FUNCTION_BLOCK ABSTRACT OpticalPowermeterBase EXTENDS TExecution IMPLEMENTS IDevice
VAR_INPUT
END_VAR
VAR_OUTPUT
END_VAR
VAR
	{attribute 'OPC.UA.DA' := '0'}
	_name : STRING;
	{attribute 'OPC.UA.DA' := '0'}
	_deviceID : STRING;					
	{attribute 'OPC.UA.DA' := '0'}
	_family : DeviceFamily;	
	{attribute 'OPC.UA.DA' := '0'}
	_logger : Logger;
	{attribute 'OPC.UA.DA' := '0'}
	_message : StringBuilder;
	{attribute 'OPC.UA.DA' := '0'}
	_opticalPowermeterConfig : DeviceConfiguration;	
END_VAR

PROPERTY DeviceID : STRING
GET
DeviceID := _deviceID;
END_GET
SET
_deviceID := DeviceID;
END_SET
END_PROPERTY

PROPERTY Family : DeviceFamily
GET
Family := _family;
END_GET
SET
_family := Family;
END_SET
END_PROPERTY

PROPERTY Name : STRING
GET
Name := _name;
END_GET
SET
_name := Name;
END_SET
END_PROPERTY

END_FUNCTION_BLOCK

(* stored: Version 1.1.0.1, ProductVersion 3.1.4024.3
   POU OpticalPowermeterBase: Id {f66f12ad-5a55-44c7-a189-9e302b9c9a12}, SpecialFunc None
   Property DeviceID: Id {e1b2634d-6751-49b6-8705-bf592686124e}
   Get Get: Id {4a34d788-a44b-4687-8c90-e0f73d1e635e}
   Set Set: Id {c660da93-b197-4dc6-80d3-da1f09d19d4c}
   Property Family: Id {7ca47322-a7a5-4a44-a085-8309d2971c79}
   Get Get: Id {4eb42a86-98bf-4e74-aca5-bf61ccc3a7ac}
   Set Set: Id {41f09890-7b88-4bb5-bbfd-19f5043d1d07}
   Property Name: Id {bac53c8c-dcd9-48c4-93a4-c6dd552b0cb6}
   Get Get: Id {c27e8b1c-eef6-41e2-b0a0-f98e58171098}
   Set Set: Id {162103b0-7c1e-4c09-874d-44c89b67e1b3} *)
